(* IEC 61131-3 sources: esstee/src/tests/programs/subrange, 2 files *)

(* ---- badrange.ST ---- *)
VAR_GLOBAL
	sr : INT(2..-10);
END_VAR

PROGRAM t

;

END_PROGRAM

(* ---- basic.ST ---- *)
VAR_GLOBAL
	sr : INT(-10..2);
	sr_default : INT(-10..2) := 2;
	sr_one : INT(1..1);
END_VAR

PROGRAM t

;

END_PROGRAM
